KUKA KRL program: chk_w9_grp3_clo.src

&ACCESS RVO1
&COMMENT Axor 903 Z3.1
DEF chk_w9_grp3_clo( )
; Check gripper AXOR 903 CLOSE Z3.1
;//---- Start User-------

$TIMER[10] = 0
$TIMER_STOP[10] = FALSE

WAIT FOR ($IN[502])
WAIT FOR (NOT $IN[501])

$TIMER_STOP[10] = TRUE
$TIMER[10] = 0

;//---- End User---------
END
